// TIA Portal project "temp" (V15)

(* hardware
DEVICE "S71500/ET200MP station_1"  S7-1500 station
   slot 0: "Rail_0"  Rack  6ES7 590-1***0-0AA0
   slot 1: "flow_control"  CPU 1512C-1 PN  6ES7 512-1CK01-0AB0  V2.5
      slot 3: "CPU display_1"  6ES7591-1AA00-0AA0
DEVICE "S7-1200 station_1"  S7-1200 Station
   slot 0: "Rack_0"  S7-1200 Rack  Rack  V1.0
   slot 1: "temperature"  CPU 1215C DC/DC/DC  6ES7 215-1AG40-0XB0  V4.0
*)

// ===== PLC "flow_control"  CPU 1512C-1 PN =====

VAR_GLOBAL   // PLC tag table "Default tag table"
   "Tag_1" AT %M0.0 : Bool;
   "Tag_2" AT %MD100 : Real;
   "Tag_3" AT %QW0 : Int;
   "Tag_4" AT %MD7 : Real;
   "Tag_5" AT %MD3 : DWord;
   "Tag_6" AT %IW0 : Int;
   "Tag_7" AT %M0.1 : Bool;
   "Tag_8" AT %M0.2 : Bool;
   "Tag_9" AT %MD11 : DWord;
   "Tag_10" AT %MD4 : Real;
   "Tag_11" AT %M0.3 : Bool;
   "Tag_12" AT %M0.6 : Bool;
END_VAR

DATA_BLOCK "Data_block_1"   // DB1
{ S7_Optimized_Access := 'FALSE' }
VERSION : 0.1
   VAR
      Kc : Real := 0.0;
      tau_i : Real := 0.0;
      tau_d : Real := 0.0;
      MVk : Real := 0.0;
      "MVk-1" : Real := 0.0;
      ek : Real := 0.0;
      "ek-1" : Real := 0.0;
      "ek-2" : Real := 0.0;
      delta_t : Real;
   END_VAR
BEGIN
END_DATA_BLOCK

FUNCTION "DAC_OUT" : Void   // FC1, LAD
{ S7_Optimized_Access := 'TRUE' }
VERSION : 0.1
   VAR_INPUT
      mv : Real;
      mv_min : Real;
      mv_max : Real;
      PQW_min : Real;
      PQW_max : Real;
   END_VAR
   VAR_OUTPUT
      PQWx : Int;
   END_VAR
   VAR_TEMP
      Temp3 : Real;
      Temp4 : Real;
      Temp5 : Real;
      Temp6 : Real;
      Temp7 : Real;
      Temp8 : Real;
   END_VAR
BEGIN

REGION Network 1
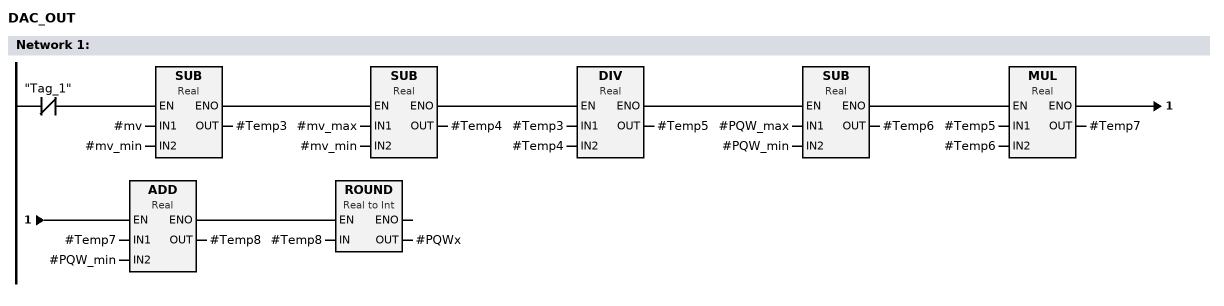
   RUNG wire#powerrail
      I_Contact( "Tag_1" )
      { S7_Templates := "SrcType := Real" } Sub(in1 := #mv, in2 := #mv_min, out => #Temp3)
      { S7_Templates := "SrcType := Real" } Sub(in1 := #mv_max, in2 := #mv_min, out => #Temp4)
      { S7_Templates := "SrcType := Real" } Div(in1 := #Temp3, in2 := #Temp4, out => #Temp5)
      { S7_Templates := "SrcType := Real" } Sub(in1 := #PQW_max, in2 := #PQW_min, out => #Temp6)
      { S7_Templates := "SrcType := Real" } Mul(in1 := #Temp5, in2 := #Temp6, out => #Temp7)
      { S7_Templates := "SrcType := Real" } Add(in1 := #Temp7, in2 := #PQW_min, out => #Temp8)
      { S7_Templates := "[SrcType := Real, DestType := Int]" } Round(in := #Temp8, out => #PQWx)
   END_RUNG
   // the same network as SCL:
   IF NOT "Tag_1" THEN
       #Temp3 := #mv - #mv_min;
       #Temp4 := #mv_max - #mv_min;
       #Temp5 := #Temp3 / #Temp4;
       #Temp6 := #PQW_max - #PQW_min;
       #Temp7 := #Temp5 * #Temp6;
       #Temp8 := #Temp7 + #PQW_min;
       #PQWx := ROUND(#Temp8);
   END_IF;
END_REGION
END_FUNCTION

FUNCTION "ADC_IN" : Void   // FC2, LAD
{ S7_Optimized_Access := 'TRUE' }
VERSION : 0.1
   VAR_INPUT
      In : Int;
   END_VAR
   VAR_OUTPUT
      Out : Real;
   END_VAR
   VAR_TEMP
      Temp1 : DInt;
      Temp2 : Real;
      Temp3 : Real;
      Temp4 : Real;
      Temp5 : Real;
      Temp6 : Real;
      Temp7 : Real;
      Temp8 : Real;
   END_VAR
   VAR CONSTANT
      PIW_max : Real := 27648.0;
      PIW_min : Real := 0.0;
      x_max : Real := 10.0;
      x_min : Real := 0.0;
   END_VAR
BEGIN

REGION Network 1
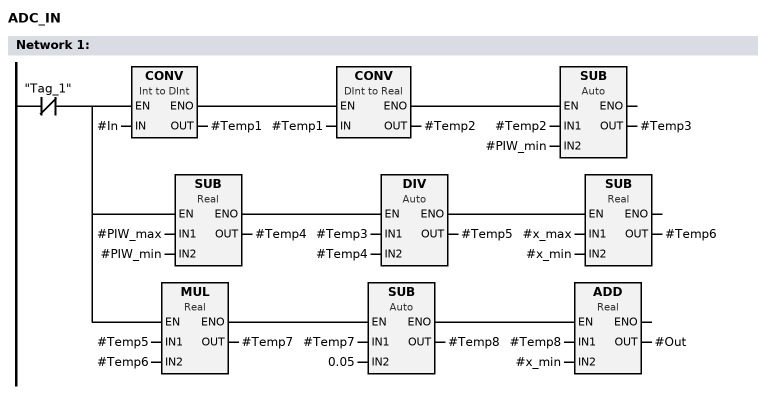
   RUNG wire#powerrail
      I_Contact( "Tag_1" )
      wire#w1
      { S7_Templates := "[SrcType := Int, DestType := DInt]" } Convert(in := #In, out => #Temp1)
      { S7_Templates := "[SrcType := DInt, DestType := Real]" } Convert(in := #Temp1, out => #Temp2)
      Sub(in1 := #Temp2, in2 := #PIW_min, out => #Temp3)
   END_RUNG
   RUNG wire#w1
      { S7_Templates := "SrcType := Real" } Sub(in1 := #PIW_max, in2 := #PIW_min, out => #Temp4)
      Div(in1 := #Temp3, in2 := #Temp4, out => #Temp5)
      { S7_Templates := "SrcType := Real" } Sub(in1 := #x_max, in2 := #x_min, out => #Temp6)
   END_RUNG
   RUNG wire#w1
      { S7_Templates := "SrcType := Real" } Mul(in1 := #Temp5, in2 := #Temp6, out => #Temp7)
      Sub(in1 := #Temp7, in2 := 0.05, out => #Temp8)
      { S7_Templates := "SrcType := Real" } Add(in1 := #Temp8, in2 := #x_min, out => #Out)
   END_RUNG
   // the same network as SCL:
   IF NOT "Tag_1" THEN
       #Temp1 := INT_TO_DINT(#In);
       #Temp2 := DINT_TO_REAL(#Temp1);
       #Temp3 := #Temp2 - #PIW_min;
       #Temp4 := #PIW_max - #PIW_min;
       #Temp5 := #Temp3 / #Temp4;
       #Temp6 := #x_max - #x_min;
       #Temp7 := #Temp5 * #Temp6;
       #Temp8 := #Temp7 - 0.05;
       #Out := #Temp8 + #x_min;
   END_IF;
END_REGION
END_FUNCTION

FUNCTION "PID" : Void   // FC3, LAD
{ S7_Optimized_Access := 'TRUE' }
VERSION : 0.1
   VAR_INPUT
      K_c : Real;
      tau_i : Real;
      tau_d : Real;
      delta_t : Real;
      "ek-1" : Real;
      "ek-2" : Real;
      ek : Real;
      "MVk-1" : Real;
   END_VAR
   VAR_OUTPUT
      MVk : Real;
      checkMV : Real;
   END_VAR
   VAR_TEMP
      Temp1 : Real;
      Temp2 : Real;
      Temp3 : Real;
      Temp4 : Real;
      Temp5 : Real;
      Temp6 : Real;
      Temp7 : Real;
      Temp8 : Real;
      Temp9 : Real;
      Temp10 : Real;
      Temp11 : Real;
      Temp12 : Real;
      Temp13 : Real;
      Temp15 : Real;
      Temp14 : Real;
      Temp16 : Real;
   END_VAR
BEGIN

REGION Network 1
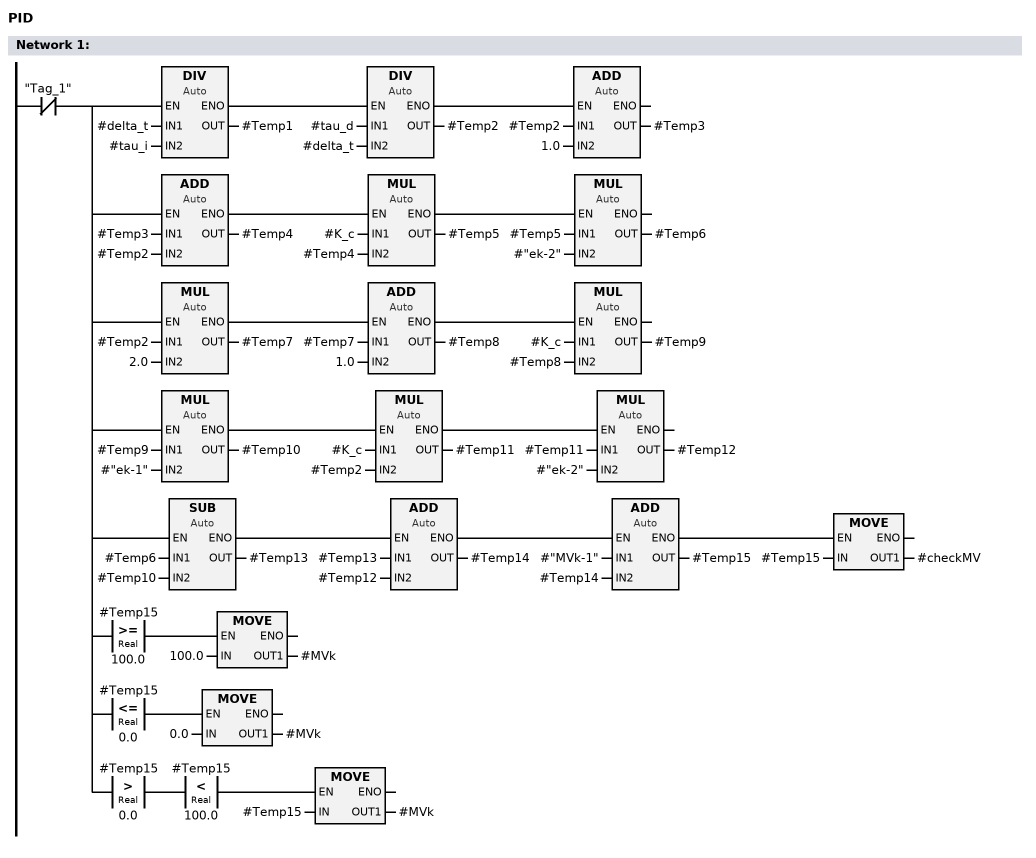
   RUNG wire#powerrail
      I_Contact( "Tag_1" )
      wire#w1
      Div(in1 := #delta_t, in2 := #tau_i, out => #Temp1)
      Div(in1 := #tau_d, in2 := #delta_t, out => #Temp2)
      Add(in1 := #Temp2, in2 := 1.0, out => #Temp3)
   END_RUNG
   RUNG wire#w1
      Add(in1 := #Temp3, in2 := #Temp2, out => #Temp4)
      Mul(in1 := #K_c, in2 := #Temp4, out => #Temp5)
      Mul(in1 := #Temp5, in2 := #"ek-2", out => #Temp6)
   END_RUNG
   RUNG wire#w1
      Mul(in1 := #Temp2, in2 := 2.0, out => #Temp7)
      Add(in1 := #Temp7, in2 := 1.0, out => #Temp8)
      Mul(in1 := #K_c, in2 := #Temp8, out => #Temp9)
   END_RUNG
   RUNG wire#w1
      Mul(in1 := #Temp9, in2 := #"ek-1", out => #Temp10)
      Mul(in1 := #K_c, in2 := #Temp2, out => #Temp11)
      Mul(in1 := #Temp11, in2 := #"ek-2", out => #Temp12)
   END_RUNG
   RUNG wire#w1
      Sub(in1 := #Temp6, in2 := #Temp10, out => #Temp13)
      Add(in1 := #Temp13, in2 := #Temp12, out => #Temp14)
      Add(in1 := #"MVk-1", in2 := #Temp14, out => #Temp15)
      Move(in := #Temp15, out1 => #checkMV)
   END_RUNG
   RUNG wire#w1
      { S7_Templates := "SrcType := Real" } GE_Contact(in1 := #Temp15, in2 := 100.0)
      Move(in := 100.0, out1 => #MVk)
   END_RUNG
   RUNG wire#w1
      { S7_Templates := "SrcType := Real" } LE_Contact(in1 := #Temp15, in2 := 0.0)
      Move(in := 0.0, out1 => #MVk)
   END_RUNG
   RUNG wire#w1
      { S7_Templates := "SrcType := Real" } GT_Contact(in1 := #Temp15, in2 := 0.0)
      { S7_Templates := "SrcType := Real" } LT_Contact(in1 := #Temp15, in2 := 100.0)
      Move(in := #Temp15, out1 => #MVk)
   END_RUNG
   // the same network as SCL:
   IF NOT "Tag_1" THEN
       #Temp1 := #delta_t / #tau_i;
       #Temp2 := #tau_d / #delta_t;
       #Temp3 := #Temp2 + 1.0;
       #Temp4 := #Temp3 + #Temp2;
       #Temp5 := #K_c * #Temp4;
       #Temp6 := #Temp5 * #"ek-2";
       #Temp7 := #Temp2 * 2.0;
       #Temp8 := #Temp7 + 1.0;
       #Temp9 := #K_c * #Temp8;
       #Temp10 := #Temp9 * #"ek-1";
       #Temp11 := #K_c * #Temp2;
       #Temp12 := #Temp11 * #"ek-2";
       #Temp13 := #Temp6 - #Temp10;
       #Temp14 := #Temp13 + #Temp12;
       #Temp15 := #"MVk-1" + #Temp14;
       #checkMV := #Temp15;
   END_IF;
   IF NOT "Tag_1" AND (#Temp15 >= 100.0) THEN #MVk := 100.0; END_IF;
   IF NOT "Tag_1" AND (#Temp15 <= 0.0) THEN #MVk := 0.0; END_IF;
   IF NOT "Tag_1" AND (#Temp15 > 0.0) AND (#Temp15 < 100.0) THEN #MVk := #Temp15; END_IF;
END_REGION
END_FUNCTION

FUNCTION "P controller" : Void   // FC4, LAD
{ S7_Optimized_Access := 'TRUE' }
VERSION : 0.1
   VAR_INPUT
      "mv_k-1" : Real;
      kc : Real;
      ek : Real;
   END_VAR
   VAR_OUTPUT
      mv_k : Real;
   END_VAR
   VAR_TEMP
      temp1 : Real;
      temp2 : Real;
   END_VAR
BEGIN

REGION Network 1
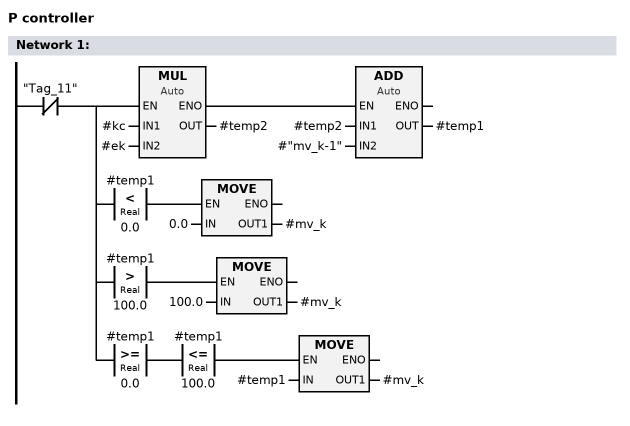
   RUNG wire#powerrail
      I_Contact( "Tag_11" )
      wire#w1
      Mul(in1 := #kc, in2 := #ek, out => #temp2)
      Add(in1 := #temp2, in2 := #"mv_k-1", out => #temp1)
   END_RUNG
   RUNG wire#w1
      { S7_Templates := "SrcType := Real" } LT_Contact(in1 := #temp1, in2 := 0.0)
      Move(in := 0.0, out1 => #mv_k)
   END_RUNG
   RUNG wire#w1
      { S7_Templates := "SrcType := Real" } GT_Contact(in1 := #temp1, in2 := 100.0)
      Move(in := 100.0, out1 => #mv_k)
   END_RUNG
   RUNG wire#w1
      { S7_Templates := "SrcType := Real" } GE_Contact(in1 := #temp1, in2 := 0.0)
      { S7_Templates := "SrcType := Real" } LE_Contact(in1 := #temp1, in2 := 100.0)
      Move(in := #temp1, out1 => #mv_k)
   END_RUNG
   // the same network as SCL:
   IF NOT "Tag_11" THEN
       #temp2 := #kc * #ek;
       #temp1 := #temp2 + #"mv_k-1";
   END_IF;
   IF NOT "Tag_11" AND (#temp1 < 0.0) THEN #mv_k := 0.0; END_IF;
   IF NOT "Tag_11" AND (#temp1 > 100.0) THEN #mv_k := 100.0; END_IF;
   IF NOT "Tag_11" AND (#temp1 >= 0.0) AND (#temp1 <= 100.0) THEN #mv_k := #temp1; END_IF;
END_REGION
END_FUNCTION

FUNCTION "PI" : Void   // FC5, LAD
{ S7_Optimized_Access := 'TRUE' }
VERSION : 0.1
   VAR_INPUT
      K_c : Real;
      tau_i : Real;
      delta_t : Real;
      "ek-1" : Real;
      ek : Real;
      "MVk-1" : Real;
   END_VAR
   VAR_OUTPUT
      mv_k : Real;
      Mv_save : Real;
   END_VAR
   VAR_TEMP
      t1 : Real;
      t2 : Real;
      t3 : Real;
      t4 : Real;
      t5 : Real;
      t6 : Real;
      t7 : Real;
      t8 : Real;
   END_VAR
BEGIN

REGION Network 1
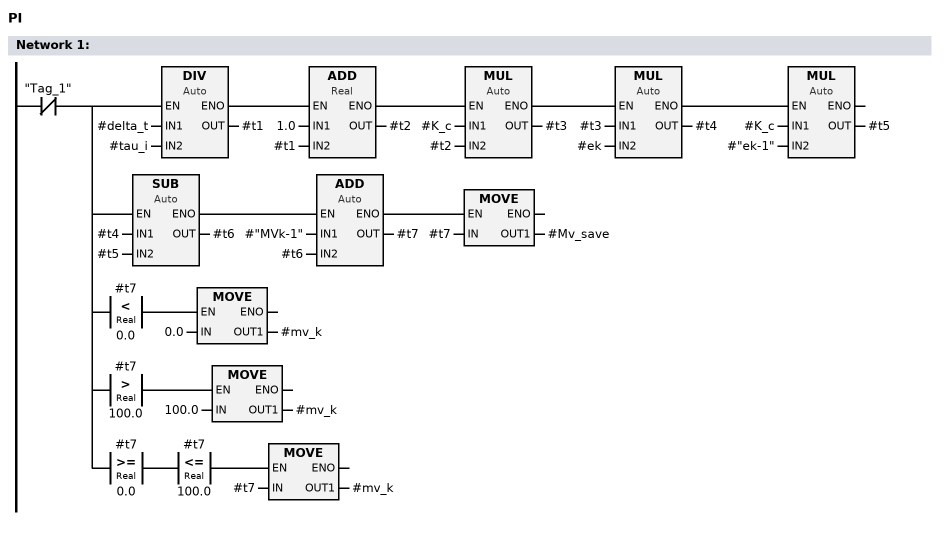
   RUNG wire#powerrail
      I_Contact( "Tag_1" )
      wire#w1
      Div(in1 := #delta_t, in2 := #tau_i, out => #t1)
      { S7_Templates := "SrcType := Real" } Add(in1 := 1.0, in2 := #t1, out => #t2)
      Mul(in1 := #K_c, in2 := #t2, out => #t3)
      Mul(in1 := #t3, in2 := #ek, out => #t4)
      Mul(in1 := #K_c, in2 := #"ek-1", out => #t5)
   END_RUNG
   RUNG wire#w1
      Sub(in1 := #t4, in2 := #t5, out => #t6)
      Add(in1 := #"MVk-1", in2 := #t6, out => #t7)
      Move(in := #t7, out1 => #Mv_save)
   END_RUNG
   RUNG wire#w1
      { S7_Templates := "SrcType := Real" } LT_Contact(in1 := #t7, in2 := 0.0)
      Move(in := 0.0, out1 => #mv_k)
   END_RUNG
   RUNG wire#w1
      { S7_Templates := "SrcType := Real" } GT_Contact(in1 := #t7, in2 := 100.0)
      Move(in := 100.0, out1 => #mv_k)
   END_RUNG
   RUNG wire#w1
      { S7_Templates := "SrcType := Real" } GE_Contact(in1 := #t7, in2 := 0.0)
      { S7_Templates := "SrcType := Real" } LE_Contact(in1 := #t7, in2 := 100.0)
      Move(in := #t7, out1 => #mv_k)
   END_RUNG
   // the same network as SCL:
   IF NOT "Tag_1" THEN
       #t1 := #delta_t / #tau_i;
       #t2 := 1.0 + #t1;
       #t3 := #K_c * #t2;
       #t4 := #t3 * #ek;
       #t5 := #K_c * #"ek-1";
       #t6 := #t4 - #t5;
       #t7 := #"MVk-1" + #t6;
       #Mv_save := #t7;
   END_IF;
   IF NOT "Tag_1" AND (#t7 < 0.0) THEN #mv_k := 0.0; END_IF;
   IF NOT "Tag_1" AND (#t7 > 100.0) THEN #mv_k := 100.0; END_IF;
   IF NOT "Tag_1" AND (#t7 >= 0.0) AND (#t7 <= 100.0) THEN #mv_k := #t7; END_IF;
END_REGION
END_FUNCTION

ORGANIZATION_BLOCK "Main"   // OB1, LAD, ProgramCycle
TITLE = "Main Program Sweep (Cycle)"
{ S7_Optimized_Access := 'TRUE' }
VERSION : 0.1
   VAR_INPUT
      Initial_Call : Bool;   // Initial call of this OB
      Remanence : Bool;   // =True, if remanent data are available
   END_VAR
   VAR_TEMP   // added for the SCL form of the ladder/FBD networks
      _w1 : Bool;
   END_VAR
BEGIN

REGION Network 1
   // Gọi hàm xác định mức chất lỏng trong bồn, MD3 là ô nhớ chứa mức lỏng trong bồn
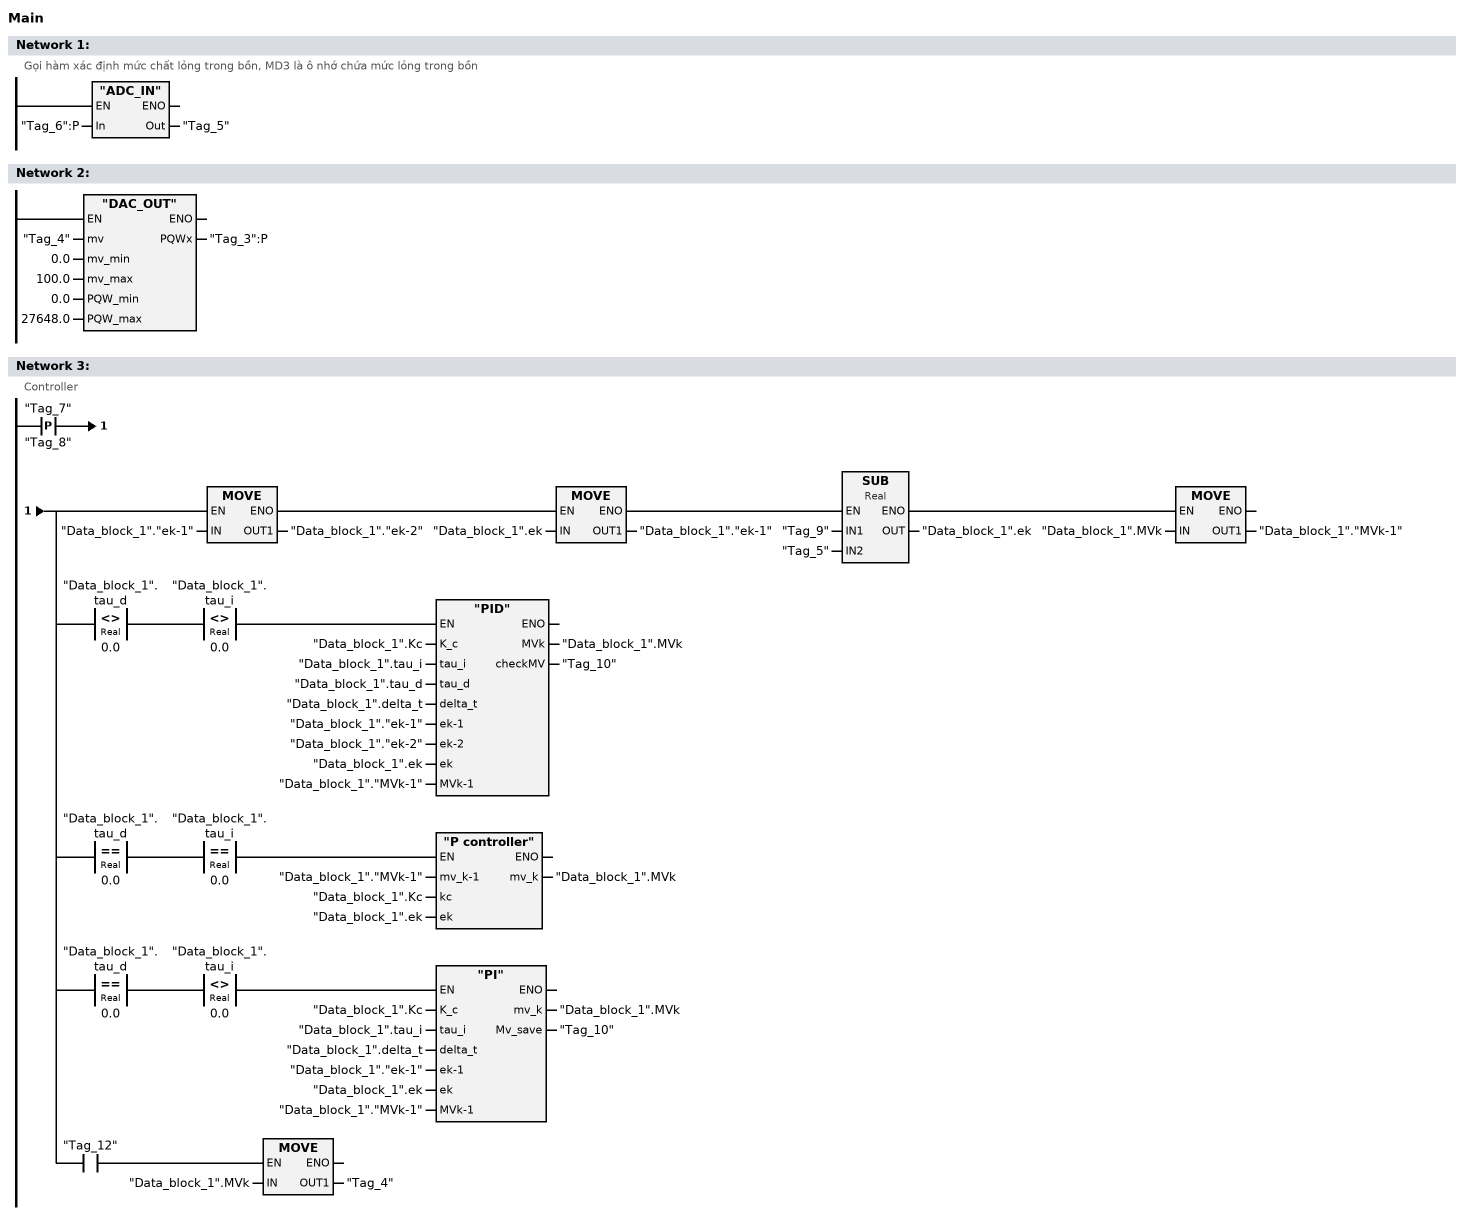
   RUNG wire#powerrail
      "ADC_IN"(In := "Tag_6":P, Out => "Tag_5")
   END_RUNG
   // the same network as SCL:
   "ADC_IN"(In := "Tag_6":P, Out => "Tag_5");
END_REGION

REGION Network 2
   RUNG wire#powerrail
      "DAC_OUT"(mv := "Tag_4", mv_min := 0.0, mv_max := 100.0, PQW_min := 0.0, PQW_max := 27648.0, PQWx => "Tag_3":P)
   END_RUNG
   // the same network as SCL:
   "DAC_OUT"(mv := "Tag_4",
             mv_min := 0.0,
             mv_max := 100.0,
             PQW_min := 0.0,
             PQW_max := 27648.0,
             PQWx => "Tag_3":P);
END_REGION

REGION Network 3
   // Controller
   RUNG wire#powerrail
      P_Contact(operand := "Tag_7", bit := "Tag_8")
      wire#w1
      Move(in := "Data_block_1"."ek-1", out1 => "Data_block_1"."ek-2")
      Move(in := "Data_block_1".ek, out1 => "Data_block_1"."ek-1")
      { S7_Templates := "SrcType := Real" } Sub(in1 := "Tag_9", in2 := "Tag_5", out => "Data_block_1".ek)
      Move(in := "Data_block_1".MVk, out1 => "Data_block_1"."MVk-1")
   END_RUNG
   RUNG wire#w1
      { S7_Templates := "SrcType := Real" } NE_Contact(in1 := "Data_block_1".tau_d, in2 := 0.0)
      { S7_Templates := "SrcType := Real" } NE_Contact(in1 := "Data_block_1".tau_i, in2 := 0.0)
      "PID"(K_c := "Data_block_1".Kc, tau_i := "Data_block_1".tau_i, tau_d := "Data_block_1".tau_d, delta_t := "Data_block_1".delta_t, "ek-1" := "Data_block_1"."ek-1", "ek-2" := "Data_block_1"."ek-2", ek := "Data_block_1".ek, "MVk-1" := "Data_block_1"."MVk-1", MVk => "Data_block_1".MVk, checkMV => "Tag_10")
   END_RUNG
   RUNG wire#w1
      { S7_Templates := "SrcType := Real" } EQ_Contact(in1 := "Data_block_1".tau_d, in2 := 0.0)
      { S7_Templates := "SrcType := Real" } EQ_Contact(in1 := "Data_block_1".tau_i, in2 := 0.0)
      "P controller"("mv_k-1" := "Data_block_1"."MVk-1", kc := "Data_block_1".Kc, ek := "Data_block_1".ek, mv_k => "Data_block_1".MVk)
   END_RUNG
   RUNG wire#w1
      { S7_Templates := "SrcType := Real" } EQ_Contact(in1 := "Data_block_1".tau_d, in2 := 0.0)
      { S7_Templates := "SrcType := Real" } NE_Contact(in1 := "Data_block_1".tau_i, in2 := 0.0)
      "PI"(K_c := "Data_block_1".Kc, tau_i := "Data_block_1".tau_i, delta_t := "Data_block_1".delta_t, "ek-1" := "Data_block_1"."ek-1", ek := "Data_block_1".ek, "MVk-1" := "Data_block_1"."MVk-1", mv_k => "Data_block_1".MVk, Mv_save => "Tag_10")
   END_RUNG
   RUNG wire#w1
      Contact( "Tag_12" )
      Move(in := "Data_block_1".MVk, out1 => "Tag_4")
   END_RUNG
   // the same network as SCL:
   #_w1 := "Tag_7" AND NOT "Tag_8";   // rising edge of "Tag_7"
   "Tag_8" := "Tag_7";
   IF #_w1 THEN
       "Data_block_1"."ek-2" := "Data_block_1"."ek-1";
       "Data_block_1"."ek-1" := "Data_block_1".ek;
       "Data_block_1".ek := "Tag_9" - "Tag_5";
       "Data_block_1"."MVk-1" := "Data_block_1".MVk;
   END_IF;
   IF #_w1 AND ("Data_block_1".tau_d <> 0.0) AND ("Data_block_1".tau_i <> 0.0) THEN
       "PID"(K_c := "Data_block_1".Kc,
             tau_i := "Data_block_1".tau_i,
             tau_d := "Data_block_1".tau_d,
             delta_t := "Data_block_1".delta_t,
             "ek-1" := "Data_block_1"."ek-1",
             "ek-2" := "Data_block_1"."ek-2",
             ek := "Data_block_1".ek,
             "MVk-1" := "Data_block_1"."MVk-1",
             MVk => "Data_block_1".MVk,
             checkMV => "Tag_10");
   END_IF;
   IF #_w1 AND ("Data_block_1".tau_d = 0.0) AND ("Data_block_1".tau_i = 0.0) THEN
       "P controller"("mv_k-1" := "Data_block_1"."MVk-1",
                      kc := "Data_block_1".Kc,
                      ek := "Data_block_1".ek,
                      mv_k => "Data_block_1".MVk);
   END_IF;
   IF #_w1 AND ("Data_block_1".tau_d = 0.0) AND ("Data_block_1".tau_i <> 0.0) THEN
       "PI"(K_c := "Data_block_1".Kc,
            tau_i := "Data_block_1".tau_i,
            delta_t := "Data_block_1".delta_t,
            "ek-1" := "Data_block_1"."ek-1",
            ek := "Data_block_1".ek,
            "MVk-1" := "Data_block_1"."MVk-1",
            mv_k => "Data_block_1".MVk,
            Mv_save => "Tag_10");
   END_IF;
   IF #_w1 AND "Tag_12" THEN "Tag_4" := "Data_block_1".MVk; END_IF;
END_REGION
END_ORGANIZATION_BLOCK

ORGANIZATION_BLOCK "Cyclic interrupt"   // OB35, LAD, CyclicInterrupt
{ S7_Optimized_Access := 'TRUE' }
VERSION : 0.1
   VAR_INPUT
      Initial_Call : Bool;   // Initial call of this OB
      Event_Count : Int;   // Events discarded
   END_VAR
   VAR_TEMP
      OB35_EV_CLASS : Byte;
   END_VAR
BEGIN

REGION Network 1
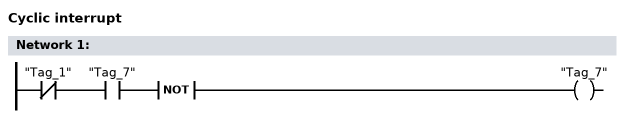
   RUNG wire#powerrail
      I_Contact( "Tag_1" )
      Contact( "Tag_7" )
      Not()
      Coil( "Tag_7" )
   END_RUNG
   // the same network as SCL:
   "Tag_7" := NOT (NOT "Tag_1" AND "Tag_7");
END_REGION
END_ORGANIZATION_BLOCK

// ===== PLC "temperature"  CPU 1215C DC/DC/DC =====

VAR_GLOBAL   // PLC tag table "Default tag table"
   "Tag_2" AT %IW64 : Int;
   "Tag_6" AT %MD3 : Real;
   "Tag_13" AT %MD7 : Real;
   "Tag_14" AT %QW64 : Int;
   "Tag_15" AT %M0.0 : Bool;
   "Tag_3" AT %M0.1 : Bool;
   "Tag_11" AT %M0.3 : Bool;
   "Tag_1" AT %MD11 : Real;
   "Tag_16" AT %M0.2 : Bool;
   "Tag_17" AT %MD4 : Real;
   "Tag_18" AT %M0.6 : Bool;
   "Tag_4" AT %MD10 : DWord;
   "Tag_5" AT %MD15 : DWord;
   "Tag_7" AT %IW66 : Int;
   "Tag_8" AT %M1.1 : Bool;
END_VAR

DATA_BLOCK "Data_block_1"   // DB1
{ S7_Optimized_Access := 'FALSE' }
VERSION : 0.1
   VAR
      Kc : Real := 0.0;
      tau_i : Real := 0.0;
      tau_d : Real := 0.0;
      MVk : Real := 0.0;
      "MVk-1" : Real := 0.0;
      ek : Real := 0.0;
      "ek-1" : Real := 0.0;
      "ek-2" : Real := 0.0;
      delta_t : Real;
   END_VAR
BEGIN
END_DATA_BLOCK

FUNCTION "DAC_OUT" : Void   // FC1, LAD
{ S7_Optimized_Access := 'TRUE' }
VERSION : 0.1
   VAR_INPUT
      mv : Real;
      mv_min : Real;
      mv_max : Real;
      PQW_min : Real;
      PQW_max : Real;
   END_VAR
   VAR_OUTPUT
      PQWx : Int;
   END_VAR
   VAR_TEMP
      Temp3 : Real;
      Temp4 : Real;
      Temp5 : Real;
      Temp6 : Real;
      Temp7 : Real;
      Temp8 : Real;
   END_VAR
BEGIN

REGION Network 1
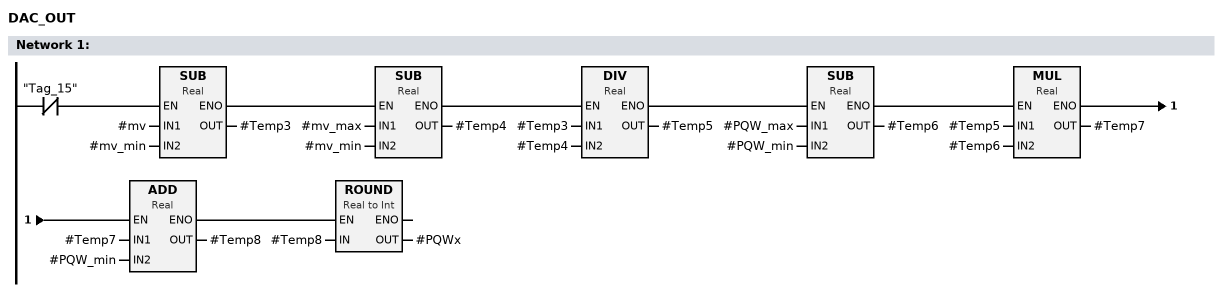
   RUNG wire#powerrail
      I_Contact( "Tag_15" )
      { S7_Templates := "SrcType := Real" } Sub(in1 := #mv, in2 := #mv_min, out => #Temp3)
      { S7_Templates := "SrcType := Real" } Sub(in1 := #mv_max, in2 := #mv_min, out => #Temp4)
      { S7_Templates := "SrcType := Real" } Div(in1 := #Temp3, in2 := #Temp4, out => #Temp5)
      { S7_Templates := "SrcType := Real" } Sub(in1 := #PQW_max, in2 := #PQW_min, out => #Temp6)
      { S7_Templates := "SrcType := Real" } Mul(in1 := #Temp5, in2 := #Temp6, out => #Temp7)
      { S7_Templates := "SrcType := Real" } Add(in1 := #Temp7, in2 := #PQW_min, out => #Temp8)
      { S7_Templates := "[SrcType := Real, DestType := Int]" } Round(in := #Temp8, out => #PQWx)
   END_RUNG
   // the same network as SCL:
   IF NOT "Tag_15" THEN
       #Temp3 := #mv - #mv_min;
       #Temp4 := #mv_max - #mv_min;
       #Temp5 := #Temp3 / #Temp4;
       #Temp6 := #PQW_max - #PQW_min;
       #Temp7 := #Temp5 * #Temp6;
       #Temp8 := #Temp7 + #PQW_min;
       #PQWx := ROUND(#Temp8);
   END_IF;
END_REGION
END_FUNCTION

FUNCTION "ADC_IN" : Void   // FC2, LAD
{ S7_Optimized_Access := 'TRUE' }
VERSION : 0.1
   VAR_INPUT
      PIW_max : Real;
      PIW_min : Real;
      x_max : Real;
      x_min : Real;
      In : Int;
   END_VAR
   VAR_OUTPUT
      Out : Real;
   END_VAR
   VAR_TEMP
      Temp1 : DInt;
      Temp2 : Real;
      Temp3 : Real;
      Temp4 : Real;
      Temp5 : Real;
      Temp6 : Real;
      Temp7 : Real;
      Temp8 : Real;
   END_VAR
BEGIN

REGION Network 1
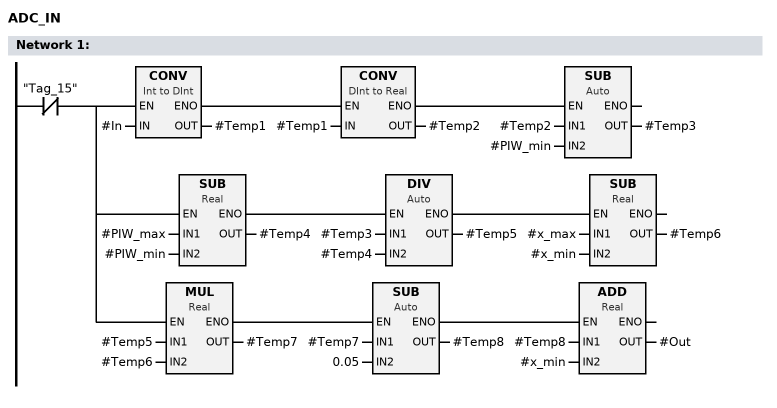
   RUNG wire#powerrail
      I_Contact( "Tag_15" )
      wire#w1
      { S7_Templates := "[SrcType := Int, DestType := DInt]" } Convert(in := #In, out => #Temp1)
      { S7_Templates := "[SrcType := DInt, DestType := Real]" } Convert(in := #Temp1, out => #Temp2)
      Sub(in1 := #Temp2, in2 := #PIW_min, out => #Temp3)
   END_RUNG
   RUNG wire#w1
      { S7_Templates := "SrcType := Real" } Sub(in1 := #PIW_max, in2 := #PIW_min, out => #Temp4)
      Div(in1 := #Temp3, in2 := #Temp4, out => #Temp5)
      { S7_Templates := "SrcType := Real" } Sub(in1 := #x_max, in2 := #x_min, out => #Temp6)
   END_RUNG
   RUNG wire#w1
      { S7_Templates := "SrcType := Real" } Mul(in1 := #Temp5, in2 := #Temp6, out => #Temp7)
      Sub(in1 := #Temp7, in2 := 0.05, out => #Temp8)
      { S7_Templates := "SrcType := Real" } Add(in1 := #Temp8, in2 := #x_min, out => #Out)
   END_RUNG
   // the same network as SCL:
   IF NOT "Tag_15" THEN
       #Temp1 := INT_TO_DINT(#In);
       #Temp2 := DINT_TO_REAL(#Temp1);
       #Temp3 := #Temp2 - #PIW_min;
       #Temp4 := #PIW_max - #PIW_min;
       #Temp5 := #Temp3 / #Temp4;
       #Temp6 := #x_max - #x_min;
       #Temp7 := #Temp5 * #Temp6;
       #Temp8 := #Temp7 - 0.05;
       #Out := #Temp8 + #x_min;
   END_IF;
END_REGION
END_FUNCTION

FUNCTION "PID" : Void   // FC3, LAD
{ S7_Optimized_Access := 'TRUE' }
VERSION : 0.1
   VAR_INPUT
      K_c : Real;
      tau_i : Real;
      tau_d : Real;
      delta_t : Real;
      "ek-1" : Real;
      "ek-2" : Real;
      ek : Real;
      "MVk-1" : Real;
   END_VAR
   VAR_OUTPUT
      MVk : Real;
      checkMV : Real;
   END_VAR
   VAR_TEMP
      Temp1 : Real;
      Temp2 : Real;
      Temp3 : Real;
      Temp4 : Real;
      Temp5 : Real;
      Temp6 : Real;
      Temp7 : Real;
      Temp8 : Real;
      Temp9 : Real;
      Temp10 : Real;
      Temp11 : Real;
      Temp12 : Real;
      Temp13 : Real;
      Temp15 : Real;
      Temp14 : Real;
      Temp16 : Real;
   END_VAR
BEGIN

REGION Network 1
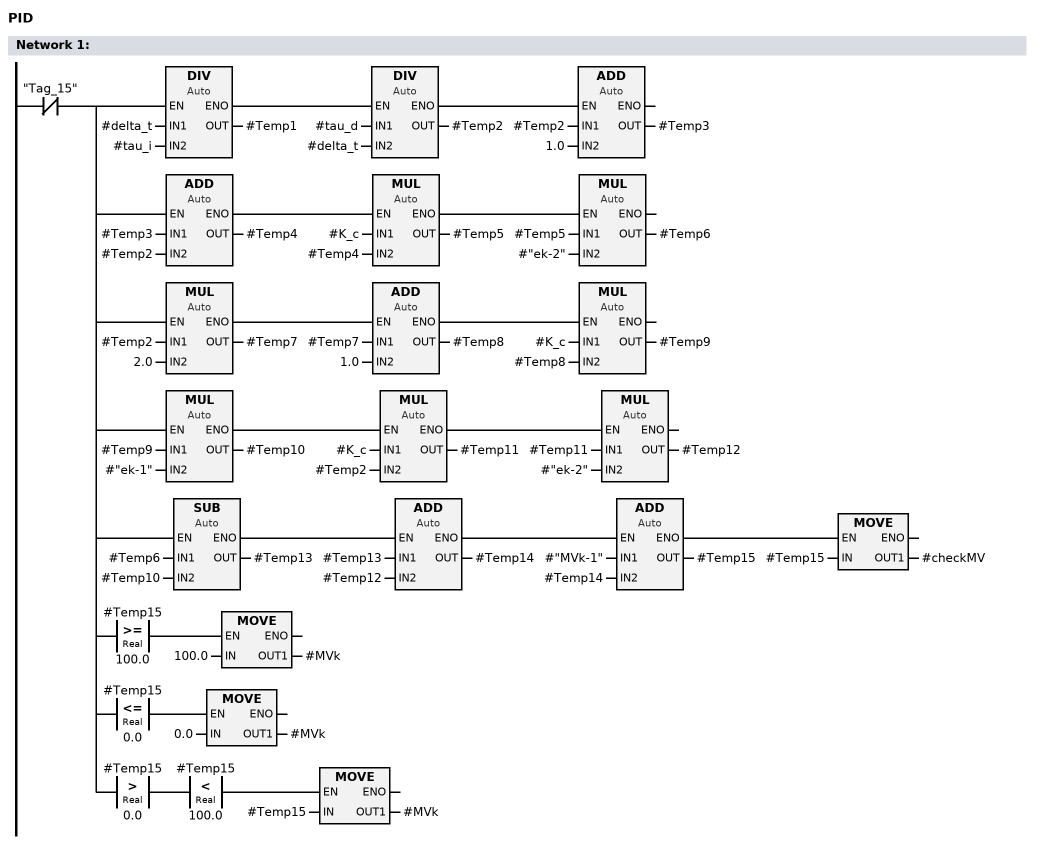
   RUNG wire#powerrail
      I_Contact( "Tag_15" )
      wire#w1
      Div(in1 := #delta_t, in2 := #tau_i, out => #Temp1)
      Div(in1 := #tau_d, in2 := #delta_t, out => #Temp2)
      Add(in1 := #Temp2, in2 := 1.0, out => #Temp3)
   END_RUNG
   RUNG wire#w1
      Add(in1 := #Temp3, in2 := #Temp2, out => #Temp4)
      Mul(in1 := #K_c, in2 := #Temp4, out => #Temp5)
      Mul(in1 := #Temp5, in2 := #"ek-2", out => #Temp6)
   END_RUNG
   RUNG wire#w1
      Mul(in1 := #Temp2, in2 := 2.0, out => #Temp7)
      Add(in1 := #Temp7, in2 := 1.0, out => #Temp8)
      Mul(in1 := #K_c, in2 := #Temp8, out => #Temp9)
   END_RUNG
   RUNG wire#w1
      Mul(in1 := #Temp9, in2 := #"ek-1", out => #Temp10)
      Mul(in1 := #K_c, in2 := #Temp2, out => #Temp11)
      Mul(in1 := #Temp11, in2 := #"ek-2", out => #Temp12)
   END_RUNG
   RUNG wire#w1
      Sub(in1 := #Temp6, in2 := #Temp10, out => #Temp13)
      Add(in1 := #Temp13, in2 := #Temp12, out => #Temp14)
      Add(in1 := #"MVk-1", in2 := #Temp14, out => #Temp15)
      Move(in := #Temp15, out1 => #checkMV)
   END_RUNG
   RUNG wire#w1
      { S7_Templates := "SrcType := Real" } GE_Contact(in1 := #Temp15, in2 := 100.0)
      Move(in := 100.0, out1 => #MVk)
   END_RUNG
   RUNG wire#w1
      { S7_Templates := "SrcType := Real" } LE_Contact(in1 := #Temp15, in2 := 0.0)
      Move(in := 0.0, out1 => #MVk)
   END_RUNG
   RUNG wire#w1
      { S7_Templates := "SrcType := Real" } GT_Contact(in1 := #Temp15, in2 := 0.0)
      { S7_Templates := "SrcType := Real" } LT_Contact(in1 := #Temp15, in2 := 100.0)
      Move(in := #Temp15, out1 => #MVk)
   END_RUNG
   // the same network as SCL:
   IF NOT "Tag_15" THEN
       #Temp1 := #delta_t / #tau_i;
       #Temp2 := #tau_d / #delta_t;
       #Temp3 := #Temp2 + 1.0;
       #Temp4 := #Temp3 + #Temp2;
       #Temp5 := #K_c * #Temp4;
       #Temp6 := #Temp5 * #"ek-2";
       #Temp7 := #Temp2 * 2.0;
       #Temp8 := #Temp7 + 1.0;
       #Temp9 := #K_c * #Temp8;
       #Temp10 := #Temp9 * #"ek-1";
       #Temp11 := #K_c * #Temp2;
       #Temp12 := #Temp11 * #"ek-2";
       #Temp13 := #Temp6 - #Temp10;
       #Temp14 := #Temp13 + #Temp12;
       #Temp15 := #"MVk-1" + #Temp14;
       #checkMV := #Temp15;
   END_IF;
   IF NOT "Tag_15" AND (#Temp15 >= 100.0) THEN #MVk := 100.0; END_IF;
   IF NOT "Tag_15" AND (#Temp15 <= 0.0) THEN #MVk := 0.0; END_IF;
   IF NOT "Tag_15" AND (#Temp15 > 0.0) AND (#Temp15 < 100.0) THEN #MVk := #Temp15; END_IF;
END_REGION
END_FUNCTION

FUNCTION "P controller" : Void   // FC4, LAD
{ S7_Optimized_Access := 'TRUE' }
VERSION : 0.1
   VAR_INPUT
      "mv_k-1" : Real;
      kc : Real;
      ek : Real;
   END_VAR
   VAR_OUTPUT
      mv_k : Real;
   END_VAR
   VAR_TEMP
      temp1 : Real;
      temp2 : Real;
   END_VAR
BEGIN

REGION Network 1
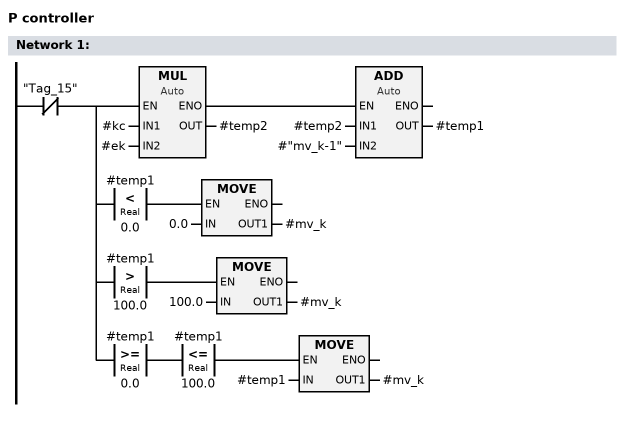
   RUNG wire#powerrail
      I_Contact( "Tag_15" )
      wire#w1
      Mul(in1 := #kc, in2 := #ek, out => #temp2)
      Add(in1 := #temp2, in2 := #"mv_k-1", out => #temp1)
   END_RUNG
   RUNG wire#w1
      { S7_Templates := "SrcType := Real" } LT_Contact(in1 := #temp1, in2 := 0.0)
      Move(in := 0.0, out1 => #mv_k)
   END_RUNG
   RUNG wire#w1
      { S7_Templates := "SrcType := Real" } GT_Contact(in1 := #temp1, in2 := 100.0)
      Move(in := 100.0, out1 => #mv_k)
   END_RUNG
   RUNG wire#w1
      { S7_Templates := "SrcType := Real" } GE_Contact(in1 := #temp1, in2 := 0.0)
      { S7_Templates := "SrcType := Real" } LE_Contact(in1 := #temp1, in2 := 100.0)
      Move(in := #temp1, out1 => #mv_k)
   END_RUNG
   // the same network as SCL:
   IF NOT "Tag_15" THEN
       #temp2 := #kc * #ek;
       #temp1 := #temp2 + #"mv_k-1";
   END_IF;
   IF NOT "Tag_15" AND (#temp1 < 0.0) THEN #mv_k := 0.0; END_IF;
   IF NOT "Tag_15" AND (#temp1 > 100.0) THEN #mv_k := 100.0; END_IF;
   IF NOT "Tag_15" AND (#temp1 >= 0.0) AND (#temp1 <= 100.0) THEN #mv_k := #temp1; END_IF;
END_REGION
END_FUNCTION

FUNCTION "PI" : Void   // FC5, LAD
{ S7_Optimized_Access := 'TRUE' }
VERSION : 0.1
   VAR_INPUT
      K_c : Real;
      tau_i : Real;
      delta_t : Real;
      "ek-1" : Real;
      ek : Real;
      "MVk-1" : Real;
   END_VAR
   VAR_OUTPUT
      mv_k : Real;
      Mv_save : Real;
   END_VAR
   VAR_TEMP
      t1 : Real;
      t2 : Real;
      t3 : Real;
      t4 : Real;
      t5 : Real;
      t6 : Real;
      t7 : Real;
      t8 : Real;
   END_VAR
BEGIN

REGION Network 1
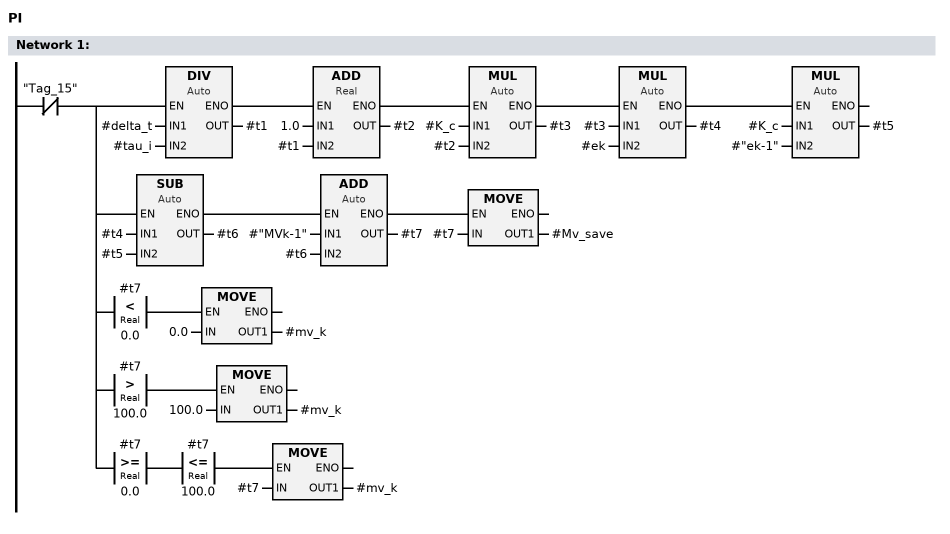
   RUNG wire#powerrail
      I_Contact( "Tag_15" )
      wire#w1
      Div(in1 := #delta_t, in2 := #tau_i, out => #t1)
      { S7_Templates := "SrcType := Real" } Add(in1 := 1.0, in2 := #t1, out => #t2)
      Mul(in1 := #K_c, in2 := #t2, out => #t3)
      Mul(in1 := #t3, in2 := #ek, out => #t4)
      Mul(in1 := #K_c, in2 := #"ek-1", out => #t5)
   END_RUNG
   RUNG wire#w1
      Sub(in1 := #t4, in2 := #t5, out => #t6)
      Add(in1 := #"MVk-1", in2 := #t6, out => #t7)
      Move(in := #t7, out1 => #Mv_save)
   END_RUNG
   RUNG wire#w1
      { S7_Templates := "SrcType := Real" } LT_Contact(in1 := #t7, in2 := 0.0)
      Move(in := 0.0, out1 => #mv_k)
   END_RUNG
   RUNG wire#w1
      { S7_Templates := "SrcType := Real" } GT_Contact(in1 := #t7, in2 := 100.0)
      Move(in := 100.0, out1 => #mv_k)
   END_RUNG
   RUNG wire#w1
      { S7_Templates := "SrcType := Real" } GE_Contact(in1 := #t7, in2 := 0.0)
      { S7_Templates := "SrcType := Real" } LE_Contact(in1 := #t7, in2 := 100.0)
      Move(in := #t7, out1 => #mv_k)
   END_RUNG
   // the same network as SCL:
   IF NOT "Tag_15" THEN
       #t1 := #delta_t / #tau_i;
       #t2 := 1.0 + #t1;
       #t3 := #K_c * #t2;
       #t4 := #t3 * #ek;
       #t5 := #K_c * #"ek-1";
       #t6 := #t4 - #t5;
       #t7 := #"MVk-1" + #t6;
       #Mv_save := #t7;
   END_IF;
   IF NOT "Tag_15" AND (#t7 < 0.0) THEN #mv_k := 0.0; END_IF;
   IF NOT "Tag_15" AND (#t7 > 100.0) THEN #mv_k := 100.0; END_IF;
   IF NOT "Tag_15" AND (#t7 >= 0.0) AND (#t7 <= 100.0) THEN #mv_k := #t7; END_IF;
END_REGION
END_FUNCTION

ORGANIZATION_BLOCK "Main"   // OB1, LAD, ProgramCycle
TITLE = "Main Program Sweep (Cycle)"
{ S7_Optimized_Access := 'TRUE' }
VERSION : 0.1
   VAR_INPUT
      Initial_Call : Bool;   // Initial call of this OB
      Remanence : Bool;   // =True, if remanent data are available
   END_VAR
   VAR_TEMP   // added for the SCL form of the ladder/FBD networks
      _w1 : Bool;
   END_VAR
BEGIN

REGION Network 1
   // Gọi hàm xác định mức chất lỏng trong bồn, MD3 là ô nhớ chứa mức lỏng trong bồn
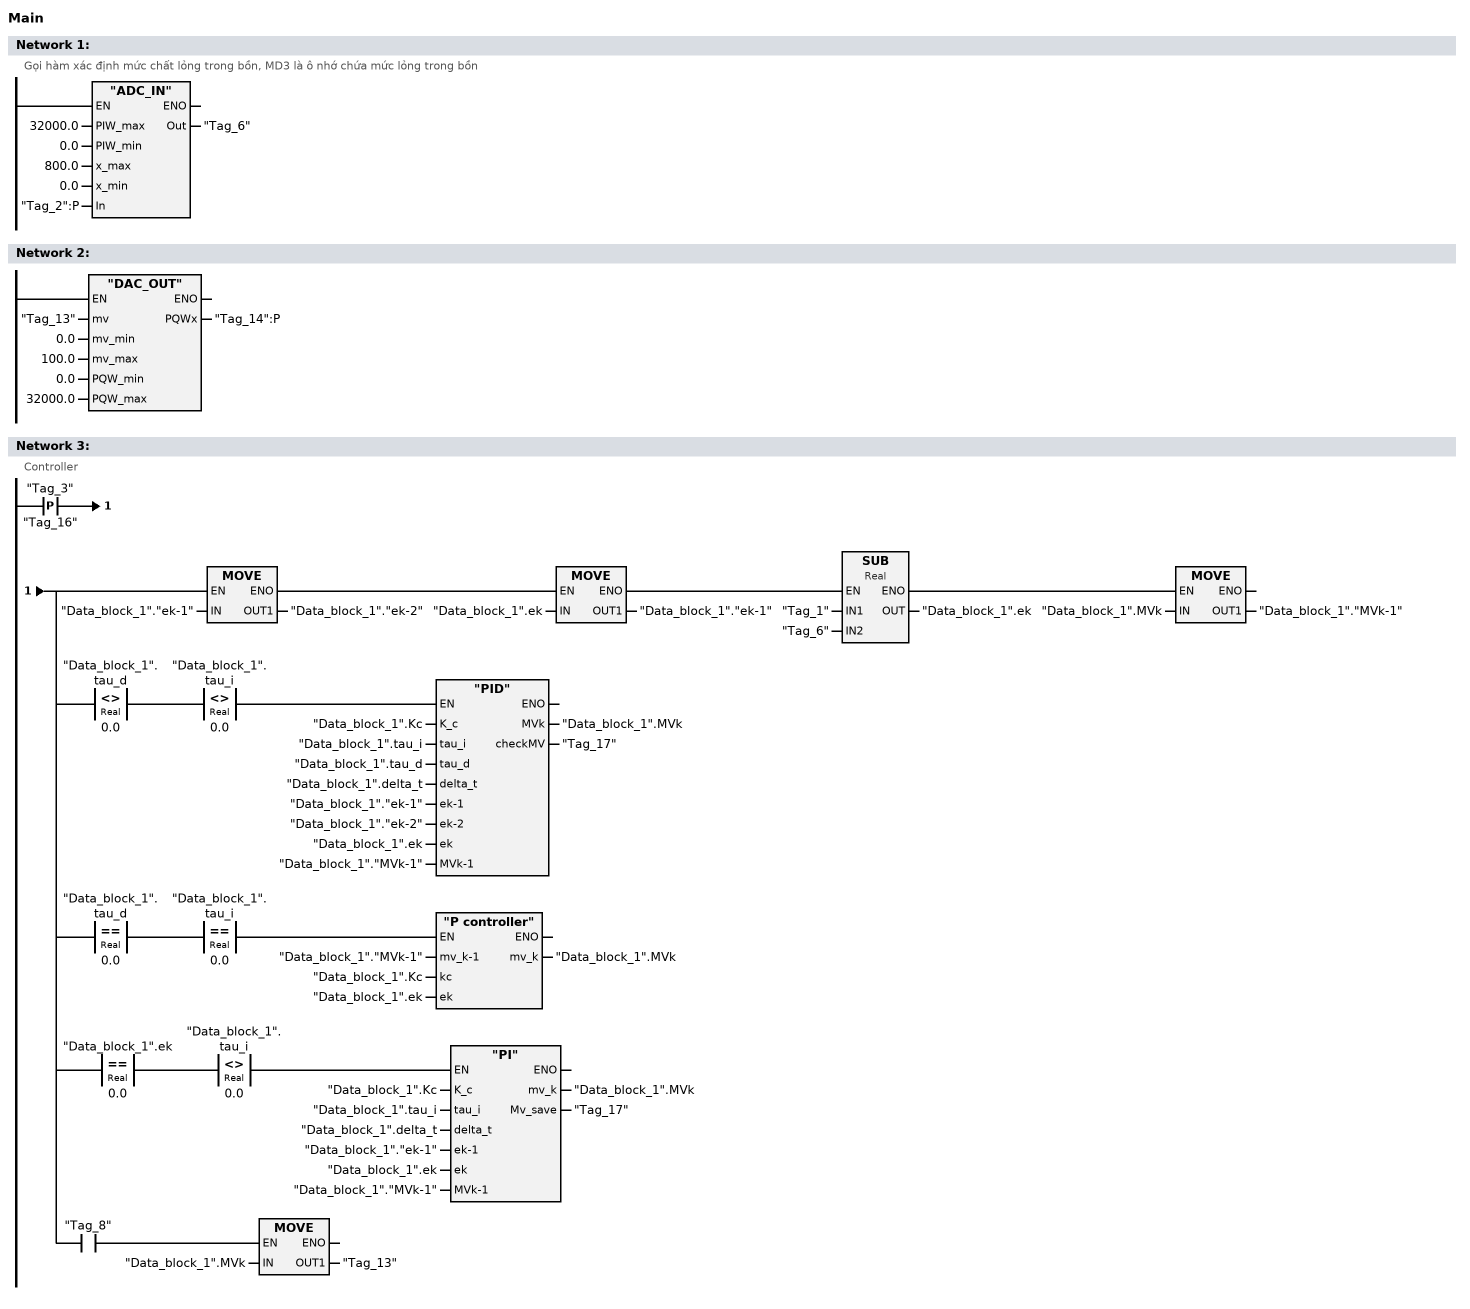
   RUNG wire#powerrail
      "ADC_IN"(PIW_max := 32000.0, PIW_min := 0.0, x_max := 800.0, x_min := 0.0, In := "Tag_2":P, Out => "Tag_6")
   END_RUNG
   // the same network as SCL:
   "ADC_IN"(PIW_max := 32000.0, PIW_min := 0.0, x_max := 800.0, x_min := 0.0, In := "Tag_2":P, Out => "Tag_6");
END_REGION

REGION Network 2
   RUNG wire#powerrail
      "DAC_OUT"(mv := "Tag_13", mv_min := 0.0, mv_max := 100.0, PQW_min := 0.0, PQW_max := 32000.0, PQWx => "Tag_14":P)
   END_RUNG
   // the same network as SCL:
   "DAC_OUT"(mv := "Tag_13",
             mv_min := 0.0,
             mv_max := 100.0,
             PQW_min := 0.0,
             PQW_max := 32000.0,
             PQWx => "Tag_14":P);
END_REGION

REGION Network 3
   // Controller
   RUNG wire#powerrail
      P_Contact(operand := "Tag_3", bit := "Tag_16")
      wire#w1
      Move(in := "Data_block_1"."ek-1", out1 => "Data_block_1"."ek-2")
      Move(in := "Data_block_1".ek, out1 => "Data_block_1"."ek-1")
      { S7_Templates := "SrcType := Real" } Sub(in1 := "Tag_1", in2 := "Tag_6", out => "Data_block_1".ek)
      Move(in := "Data_block_1".MVk, out1 => "Data_block_1"."MVk-1")
   END_RUNG
   RUNG wire#w1
      { S7_Templates := "SrcType := Real" } NE_Contact(in1 := "Data_block_1".tau_d, in2 := 0.0)
      { S7_Templates := "SrcType := Real" } NE_Contact(in1 := "Data_block_1".tau_i, in2 := 0.0)
      "PID"(K_c := "Data_block_1".Kc, tau_i := "Data_block_1".tau_i, tau_d := "Data_block_1".tau_d, delta_t := "Data_block_1".delta_t, "ek-1" := "Data_block_1"."ek-1", "ek-2" := "Data_block_1"."ek-2", ek := "Data_block_1".ek, "MVk-1" := "Data_block_1"."MVk-1", MVk => "Data_block_1".MVk, checkMV => "Tag_17")
   END_RUNG
   RUNG wire#w1
      { S7_Templates := "SrcType := Real" } EQ_Contact(in1 := "Data_block_1".tau_d, in2 := 0.0)
      { S7_Templates := "SrcType := Real" } EQ_Contact(in1 := "Data_block_1".tau_i, in2 := 0.0)
      "P controller"("mv_k-1" := "Data_block_1"."MVk-1", kc := "Data_block_1".Kc, ek := "Data_block_1".ek, mv_k => "Data_block_1".MVk)
   END_RUNG
   RUNG wire#w1
      { S7_Templates := "SrcType := Real" } EQ_Contact(in1 := "Data_block_1".ek, in2 := 0.0)
      { S7_Templates := "SrcType := Real" } NE_Contact(in1 := "Data_block_1".tau_i, in2 := 0.0)
      "PI"(K_c := "Data_block_1".Kc, tau_i := "Data_block_1".tau_i, delta_t := "Data_block_1".delta_t, "ek-1" := "Data_block_1"."ek-1", ek := "Data_block_1".ek, "MVk-1" := "Data_block_1"."MVk-1", mv_k => "Data_block_1".MVk, Mv_save => "Tag_17")
   END_RUNG
   RUNG wire#w1
      Contact( "Tag_8" )
      Move(in := "Data_block_1".MVk, out1 => "Tag_13")
   END_RUNG
   // the same network as SCL:
   #_w1 := "Tag_3" AND NOT "Tag_16";   // rising edge of "Tag_3"
   "Tag_16" := "Tag_3";
   IF #_w1 THEN
       "Data_block_1"."ek-2" := "Data_block_1"."ek-1";
       "Data_block_1"."ek-1" := "Data_block_1".ek;
       "Data_block_1".ek := "Tag_1" - "Tag_6";
       "Data_block_1"."MVk-1" := "Data_block_1".MVk;
   END_IF;
   IF #_w1 AND ("Data_block_1".tau_d <> 0.0) AND ("Data_block_1".tau_i <> 0.0) THEN
       "PID"(K_c := "Data_block_1".Kc,
             tau_i := "Data_block_1".tau_i,
             tau_d := "Data_block_1".tau_d,
             delta_t := "Data_block_1".delta_t,
             "ek-1" := "Data_block_1"."ek-1",
             "ek-2" := "Data_block_1"."ek-2",
             ek := "Data_block_1".ek,
             "MVk-1" := "Data_block_1"."MVk-1",
             MVk => "Data_block_1".MVk,
             checkMV => "Tag_17");
   END_IF;
   IF #_w1 AND ("Data_block_1".tau_d = 0.0) AND ("Data_block_1".tau_i = 0.0) THEN
       "P controller"("mv_k-1" := "Data_block_1"."MVk-1",
                      kc := "Data_block_1".Kc,
                      ek := "Data_block_1".ek,
                      mv_k => "Data_block_1".MVk);
   END_IF;
   IF #_w1 AND ("Data_block_1".ek = 0.0) AND ("Data_block_1".tau_i <> 0.0) THEN
       "PI"(K_c := "Data_block_1".Kc,
            tau_i := "Data_block_1".tau_i,
            delta_t := "Data_block_1".delta_t,
            "ek-1" := "Data_block_1"."ek-1",
            ek := "Data_block_1".ek,
            "MVk-1" := "Data_block_1"."MVk-1",
            mv_k => "Data_block_1".MVk,
            Mv_save => "Tag_17");
   END_IF;
   IF #_w1 AND "Tag_8" THEN "Tag_13" := "Data_block_1".MVk; END_IF;
END_REGION
END_ORGANIZATION_BLOCK

ORGANIZATION_BLOCK "Cyclic interrupt"   // OB35, LAD, CyclicInterrupt
{ S7_Optimized_Access := 'TRUE' }
VERSION : 0.1
   VAR_INPUT
      Initial_Call : Bool;   // Initial call of this OB
      Event_Count : Int;   // Events discarded
   END_VAR
   VAR_TEMP
      OB35_EV_CLASS : Byte;
   END_VAR
BEGIN

REGION Network 1
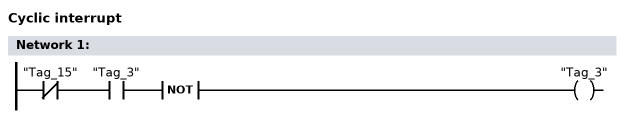
   RUNG wire#powerrail
      I_Contact( "Tag_15" )
      Contact( "Tag_3" )
      Not()
      Coil( "Tag_3" )
   END_RUNG
   // the same network as SCL:
   "Tag_3" := NOT (NOT "Tag_15" AND "Tag_3");
END_REGION
END_ORGANIZATION_BLOCK